FUNCTION_BLOCK FB_PU_St
VAR_IN_OUT
END_VAR
VAR_INPUT
END_VAR
VAR_OUTPUT
	{attribute 'OPC.UA.DA' := '1'}Zustand					: ST_PU_Zustand;	
	{attribute 'OPC.UA.DA' := '1'}Parameter				: ST_PU_Parameter;		
END_VAR
VAR
	Zustandscheck			: FB_PU_St_Zustandscheck;
END_VAR

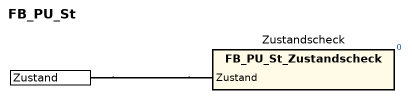
Zustandscheck(Zustand := Zustand); // FB_PU_St_Zustandscheck

END_FUNCTION_BLOCK

(* stored: Version 1.1.0.1, ProductVersion 3.1.4024.9
   POU FB_PU_St: Id {0b6b1056-4c62-4703-8bc4-8135e7b5ab79}, SpecialFunc None *)
